// TIA Portal V18 export
DATA_BLOCK "SS1_762A1_16DI_DI_Vars"   // DB11061
{ S7_Optimized_Access := 'FALSE' }
VERSION : 0.1
// stored: AutoNumber false, DBAccessibleFromOPCUA true, IsOnlyStoredInLoadMemory false, IsWriteProtectedInAS false
   VAR
      DI1 : "UDT_DIadv";   // HS Робота насосу опалення 2 (10.203)
      DI2 : "UDT_DIadv";   // Резерв
      DI3 : "UDT_DIadv";   // Резерв
      DI4 : "UDT_DIadv";   // Резерв
      DI5 : "UDT_DIadv";   // Резерв
      DI6 : "UDT_DIadv";   // Резерв
      DI7 : "UDT_DIadv";   // Резерв
      DI8 : "UDT_DIadv";   // Резерв
      DI9 { S7_SetPoint := 'True'} : "UDT_DIadv";   // Резерв
      DI10 { S7_SetPoint := 'True'} : "UDT_DIadv";   // Резерв
      DI11 { S7_SetPoint := 'True'} : "UDT_DIadv";   // Резерв
      DI12 { S7_SetPoint := 'True'} : "UDT_DIadv";   // Резерв
      DI13 { S7_SetPoint := 'True'} : "UDT_DIadv";   // Резерв
      DI14 { S7_SetPoint := 'True'} : "UDT_DIadv";   // Резерв
      DI15 { S7_SetPoint := 'True'} : "UDT_DIadv";   // Резерв
      DI16 { S7_SetPoint := 'True'} : "UDT_DIadv";   // Резерв
   END_VAR
BEGIN
   DI1.cFuncSystemID := 100;
   DI1.cFuncVar := 1;
   DI2.cFuncSystemID := 100;
   DI2.cFuncVar := 3;
   DI5.cFuncSystemID := 100;
   DI5.cFuncVar := 5;
   DI6.cFuncSystemID := 100;
   DI6.cFuncVar := 6;
END_DATA_BLOCK
